{attribute 'linkalways'} 
{attribute 'no_explicit_call' := 'This FB is a CLASS and must be accessed using methods or properties'}
{attribute 'enable_dynamic_creation'}
FUNCTION_BLOCK FINAL SEL_INT EXTENDS Node
VAR
	g : _BOOL(FALSE);
	in1 : _INT(0);
	in2 : _INT(0);
	out : _INT(0);
END_VAR

METHOD PUBLIC Clone : I_Node
VAR
	pNode : POINTER TO SEL_INT;
END_VAR
pNode := __NEW(SEL_INT);
Clone := pNode^;
END_METHOD

METHOD FB_init : BOOL
VAR_INPUT
	bInitRetains : BOOL; // if TRUE, the retain variables are initialized (warm start / cold start)
	bInCopyCode : BOOL;  // if TRUE, the instance afterwards gets moved into the copy code (online change)
END_VAR
AddInput('g',THIS^.g);
AddInput('in1',THIS^.in1);
AddInput('in2',THIS^.in2);
AddOutput('out', THIS^.out);
END_METHOD

METHOD PROTECTED OnExecute
VAR
END_VAR
IF g.value THEN
	out.value := in2.value;
ELSE
	out.value := in1.value;
END_IF
END_METHOD

END_FUNCTION_BLOCK

(* stored: Version 1.1.0.1, ProductVersion 3.1.4024.15
   POU SEL_INT: Id {767617c0-72e6-43b6-aa98-96ebcd889f69}, SpecialFunc None
   Folder Constructor: Id {75257ce6-403e-4cb0-9bbd-48b02adabd3d}
   Method Clone: Id {89e77ded-5fea-43c3-b33a-f42f90391679}
   Method FB_init: Id {94b7a816-0c53-4eb0-b483-d181dac2b270}
   Method OnExecute: Id {0ad7ff18-2e4c-4ed7-8f94-34b52e11d335} *)
